SUBAPPLICATION Uebung_206b (* Interlock: ILOCK_T_FF (Drei gegenseitig verriegelte Toggle-Flip-Flops via Adapter-Kette) *)
  (* Standard: 61499-2; Description: Copyright (c) 2026 Meisterschulen am Ostbahnhof This program and the accompanying materials are made available under the terms of the Eclipse Public License 2.0 which is available at https://www.eclipse.org/legal/epl-2.0/ SPDX-License-Identifier: EPL-2.0 *)
  (* Version 1.0, 2026-05-07, Gemini CLI, Meisterschulen am Ostbahnhof, initial version using library block ILOCK_T_FF *)
  PACKAGE Uebungen;
  IMPORT logiBUS::io::DI::logiBUS_DI::Input_I1;
  IMPORT logiBUS::io::DI::logiBUS_DI::Input_I2;
  IMPORT logiBUS::io::DI::logiBUS_DI::Input_I3;
  IMPORT logiBUS::io::DI::logiBUS_DI_Events::BUTTON_SINGLE_CLICK;
  IMPORT logiBUS::io::DQ::logiBUS_DO::Output_Q1;
  IMPORT logiBUS::io::DQ::logiBUS_DO::Output_Q2;
  IMPORT logiBUS::io::DQ::logiBUS_DO::Output_Q3;
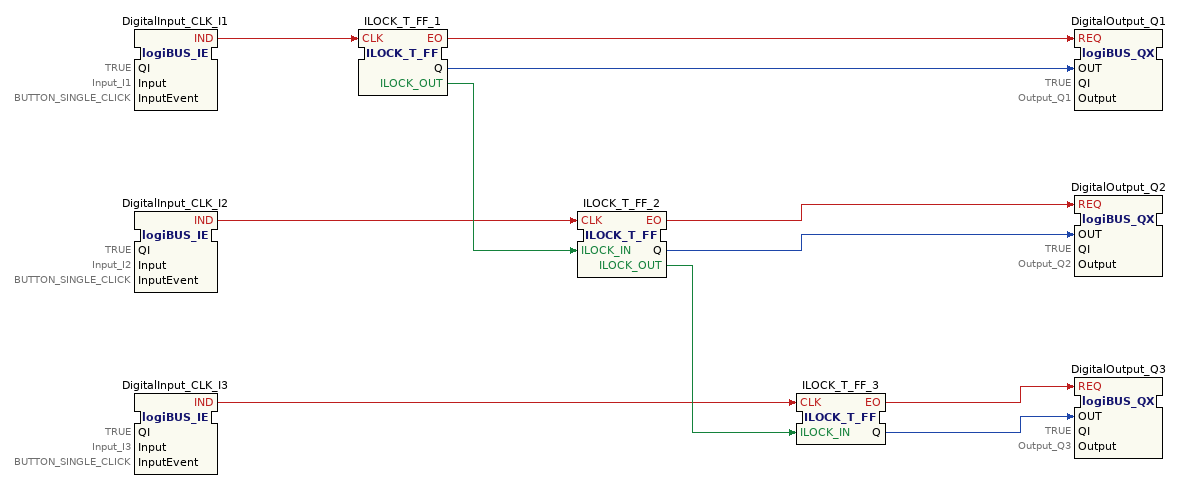
  (* Gegenseitige Verriegelung via AE2-Adapter-Kette (Bidirektional) *)
  FBS
    DigitalInput_CLK_I1 : logiBUS::io::DI::logiBUS_IE(QI := TRUE, Input := Input_I1, InputEvent := BUTTON_SINGLE_CLICK);
    DigitalInput_CLK_I2 : logiBUS::io::DI::logiBUS_IE(QI := TRUE, Input := Input_I2, InputEvent := BUTTON_SINGLE_CLICK);
    DigitalInput_CLK_I3 : logiBUS::io::DI::logiBUS_IE(QI := TRUE, Input := Input_I3, InputEvent := BUTTON_SINGLE_CLICK);
    ILOCK_T_FF_1 : logiBUS::signalprocessing::interlock::ILOCK_T_FF;
    ILOCK_T_FF_2 : logiBUS::signalprocessing::interlock::ILOCK_T_FF;
    ILOCK_T_FF_3 : logiBUS::signalprocessing::interlock::ILOCK_T_FF;
    DigitalOutput_Q1 : logiBUS::io::DQ::logiBUS_QX(QI := TRUE, Output := Output_Q1);
    DigitalOutput_Q2 : logiBUS::io::DQ::logiBUS_QX(QI := TRUE, Output := Output_Q2);
    DigitalOutput_Q3 : logiBUS::io::DQ::logiBUS_QX(QI := TRUE, Output := Output_Q3);
  END_FBS
  EVENT_CONNECTIONS
    DigitalInput_CLK_I1.IND TO ILOCK_T_FF_1.CLK;
    DigitalInput_CLK_I2.IND TO ILOCK_T_FF_2.CLK;
    DigitalInput_CLK_I3.IND TO ILOCK_T_FF_3.CLK;
    ILOCK_T_FF_1.EO TO DigitalOutput_Q1.REQ;
    ILOCK_T_FF_2.EO TO DigitalOutput_Q2.REQ;
    ILOCK_T_FF_3.EO TO DigitalOutput_Q3.REQ;
  END_CONNECTIONS
  DATA_CONNECTIONS
    ILOCK_T_FF_1.Q TO DigitalOutput_Q1.OUT;
    ILOCK_T_FF_2.Q TO DigitalOutput_Q2.OUT;
    ILOCK_T_FF_3.Q TO DigitalOutput_Q3.OUT;
  END_CONNECTIONS
  ADAPTER_CONNECTIONS
    ILOCK_T_FF_1.ILOCK_OUT TO ILOCK_T_FF_2.ILOCK_IN;
    ILOCK_T_FF_2.ILOCK_OUT TO ILOCK_T_FF_3.ILOCK_IN;
  END_CONNECTIONS
END_SUBAPPLICATION
